// TIA Portal V17 export
// export: Created 2024-08-20T13:26:08.9627556Z, ExportSetting WithDefaults, DisplayName Totally Integrated Automation Portal, DisplayVersion V17 Update 4, DisplayName TIA Portal Openness, DisplayVersion V17 Update 4, DisplayName TIA Portal Version Control Interface, DisplayVersion V17, DisplayName STEP 7 Professional, DisplayVersion V17 Update 4, DisplayName STEP 7 Safety, DisplayVersion V17, DisplayName WinCC Advanced, DisplayVersion V17 Update 4
ORGANIZATION_BLOCK "Main"   // OB1, LAD, ProgramCycle
TITLE = "Main Program Sweep (Cycle)"
{ S7_Optimized_Access := 'TRUE' }
VERSION : 0.1
// stored: AutoNumber true, IsIECCheckEnabled false, SetENOAutomatically false
   VAR_INPUT
      Initial_Call : Bool;   // Initial call of this OB
      Remanence : Bool;   // =True, if remanent data are available
   END_VAR
BEGIN

REGION Network 1: PULSO 1 SEGUNDO
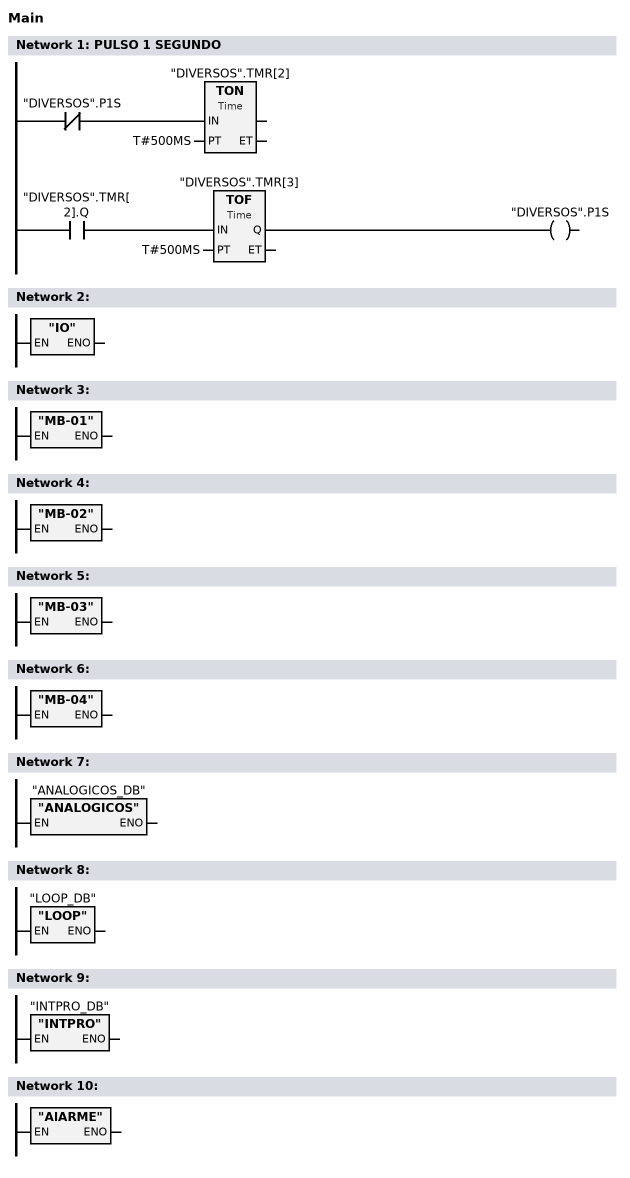
   RUNG wire#powerrail
      I_Contact( "DIVERSOS".P1S )
      { S7_Templates := "time_type := Time" } "DIVERSOS".TMR[2].TON(pt := T#500MS, et =>)
   END_RUNG
   RUNG wire#powerrail
      Contact( "DIVERSOS".TMR[2].Q )
      { S7_Templates := "time_type := Time" } "DIVERSOS".TMR[3].TOF(pt := T#500MS, et =>)
      Coil( "DIVERSOS".P1S )
   END_RUNG
   // the same network as SCL:
   "DIVERSOS".TMR[2].TON(IN := NOT "DIVERSOS".P1S, PT := T#500MS);
   "DIVERSOS".TMR[3].TOF(IN := "DIVERSOS".TMR[2].Q, PT := T#500MS);
   "DIVERSOS".P1S := "DIVERSOS".TMR[3].Q;
END_REGION

REGION Network 2
   RUNG wire#powerrail
      "IO"()
   END_RUNG
   // the same network as SCL:
   "IO"();
END_REGION

REGION Network 3
   RUNG wire#powerrail
      "MB-01"()
   END_RUNG
   // the same network as SCL:
   "MB-01"();
END_REGION

REGION Network 4
   RUNG wire#powerrail
      "MB-02"()
   END_RUNG
   // the same network as SCL:
   "MB-02"();
END_REGION

REGION Network 5
   RUNG wire#powerrail
      "MB-03"()
   END_RUNG
   // the same network as SCL:
   "MB-03"();
END_REGION

REGION Network 6
   RUNG wire#powerrail
      "MB-04"()
   END_RUNG
   // the same network as SCL:
   "MB-04"();
END_REGION

REGION Network 7
   RUNG wire#powerrail
      "ANALOGICOS_DB"()
   END_RUNG
   // the same network as SCL:
   "ANALOGICOS_DB"();   // "ANALOGICOS"
END_REGION

REGION Network 8
   RUNG wire#powerrail
      "LOOP_DB"()
   END_RUNG
   // the same network as SCL:
   "LOOP_DB"();   // "LOOP"
END_REGION

REGION Network 9
   RUNG wire#powerrail
      "INTPRO_DB"()
   END_RUNG
   // the same network as SCL:
   "INTPRO_DB"();   // "INTPRO"
END_REGION

REGION Network 10
   RUNG wire#powerrail
      "AlARME"()
   END_RUNG
   // the same network as SCL:
   "AlARME"();
END_REGION
END_ORGANIZATION_BLOCK
